// TIA Portal V21 export
TYPE "MotorPos_CFG_Type"
   STRUCT
      "xmm/degree" { S7_SetPoint := 'True'} : Bool;   // UM= Millimetri UNM= Gradi
      "xCurveS-L" { S7_SetPoint := 'True'} : Int;   // 0=curva TRAPEZIO 1=curva LOGARITMO 2=curva COS
      fJogSpeed { S7_SetPoint := 'True'} : Real := 10.0;   // Speed Jog movement (mm/sec) / Velocità JOG (mm/sec)
      fJogAcc { S7_SetPoint := 'True'} : Real := 10.0;   // Acc. jog movement (mm/sec^2) / Acc. JOG (mm/sec^2)
      fJogDec { S7_SetPoint := 'True'} : Real := 10.0;   // Dec. jog movement (mm/sec^2) / Dec. JOG (mm/sec^2)
      fVirtEncWindPos { S7_SetPoint := 'True'} : Real := 1.0;   // Cycle end virtual encoder position window (mm) / Finestra di posizione encoder virtuale Stop (mm)
      fVirtEncWindSpeed { S7_SetPoint := 'True'} : Real := 10.0;   // Cycle end virtual encoder speed window(mm/sec) / Finestra di velocità encoder virtuale Stop (mm/sec)
      fMotWindPos { S7_SetPoint := 'True'} : Real := 1.0;   // Cycle end motor position window (mm) / Finestra di posizione motore Stop (mm)
      fMotWindSpeed { S7_SetPoint := 'True'} : Real := 10.0;   // Cycle end motor speed window (mm/sec) / Finestra di velocità motore Stop (mm/sec)
      fMotAdvStopPosition { S7_SetPoint := 'True'} : Real;   // Finestra per anticipo STOP al target virtuale
      fMaxErrEnc { S7_SetPoint := 'True'} : Real := 5.0;   // Max tracking value for alarm (mm) / Massimo valore inseguimento per allarme (mm)
      fKPpid_Pos { S7_SetPoint := 'True'} : Real := 1.0;   // PID Proportional constant / Anello Posizione Costante proporzionale PID
      fKPpidAcc_Pos { S7_SetPoint := 'True'} : Real := 1.0;   // Anello Posizione Costante proporzionale PID fase accelerazione
      fKPpidDec_Pos { S7_SetPoint := 'True'} : Real := 4.0;   // PID Proportional constant dec.phase / Anello Posizione Costante proporzionale PID fase decelerazione
      fKPpid_Vel { S7_SetPoint := 'True'} : Real := 1.0;   // Anello Velocità Costante proporzionale PID
      fKPpidAcc_Vel { S7_SetPoint := 'True'} : Real := 1.0;   // Anello Velocità Costante proporzionale PID fase accelerazione
      fKPpidDec_Vel { S7_SetPoint := 'True'} : Real := 1.0;   // Anello Velocità Costante proporzionale PID fase decelerazione
      fMinSpeed { S7_SetPoint := 'True'} : Real;   // Low limit speed requested (mm/sec) / Limite INF velocità richiesta (mm/sec)
      fMaxSpeed { S7_SetPoint := 'True'} : Real := 100.0;   // High speed limit (mm/sec) / Limite SUP velocità richiesta (mm/sec)
      fFirstStepNepero { S7_SetPoint := 'True'} : Real := 6.0;   // Definisce gradino di ingresso Funzione Nepero
      "fAutoChangeS-Lvalue" { S7_SetPoint := 'True'} : Real;   // Cambio curva automatico se LOG -> TRA per spostamenti inferiori a...
      dnTimerStopEnable { S7_SetPoint := 'True'} : DInt := DINT#300;   // Value timer run inverter request (mS) / Valore timer stop richiesta marcia (mS)
      dnTimerStopEndPos { S7_SetPoint := 'True'} : DInt := DINT#1000;   // Value timer alarm positioner / Valore timer allarme controllo fine posizionamento
      dnTimerStartEnableBrake { S7_SetPoint := 'True'} : DInt := DINT#300;   // Value timer alarm positioner / Valore timer sblocco freno salita
   END_STRUCT;
END_TYPE
